// TIA Portal V19 export
DATA_BLOCK "ABFV 201 FEED BACK FLUSH"   // DB175
// stored: InstanceOfName FLUSHING VALVE, InstanceOfType FB
"FLUSHING VALVE"
   // VAR_INPUT
   //    "SUBOUTPUT VALVE" : Bool;
   //    "OPEN FEEDBACK" : Bool;
   //    "CLOSE FEEDBACK" : Bool;
   // END_VAR
   // VAR_OUTPUT
   //    "OPEN OUTPUT VAVLE" : Bool;
   //    "CLOSE OUTPUT VAVLE" : Bool;
   // END_VAR
   // VAR
   //    TIMER_1 { S7_SetPoint := 'True'} : TON_TIME;
   //    "TIMER" { S7_SetPoint := 'True'} : TON_TIME;
   // END_VAR
BEGIN
END_DATA_BLOCK
